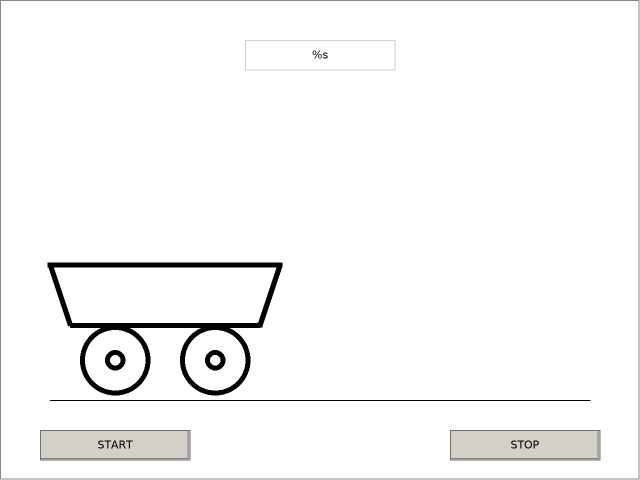
VISUALIZATION Visualization  // 640x480
    Line (50,400) (590,400)
    Group (50,265 230x130)
        p3560616238: MAIN.Visualization.Position
        Ellipse (30,60 70x70)
        Ellipse (55,85 20x20)
        Ellipse (130,60 70x70)
        Ellipse (155,85 20x20)
        Polyline (20,60) (210,60) (230,0) (0,0) (20,60)
    Button (40,430 150x30), "START"
        tap GVL.bStart
    Button (450,430 150x30), "STOP"
        tap GVL.bStop
    Textfield (245,40 150x30), "%s", text variable: MAIN.StateMachine.sState
END_VISUALIZATION

(* stored: Version 1.1.0.1, ProductVersion 3.1.4024.12
   Visu Visualization: Id {c703bc2b-e8ba-4143-ac38-3a1635d144b4} *)
